FUNCTION_BLOCK LIntComparer EXTENDS Object IMPLEMENTS IComparer
VAR
	_ClassName : STRING := __POUNAME();
END_VAR

{attribute 'monitoring' := 'call'}
PROPERTY ClassName : STRING
GET
ClassName := _ClassName;
END_GET
END_PROPERTY

{attribute "object_name" := "Compare"}
METHOD Compare : COMPARISION_RESULT
VAR_INPUT
	left : __SYSTEM.AnyType;
	right : __SYSTEM.AnyType;
END_VAR
VAR
	leftPointer : POINTER TO LINT; 
	rightPointer : POINTER TO LINT; 
END_VAR
IF left.pValue = 0 AND right.pValue = 0 THEN
	Compare := COMPARISION_RESULT.FIRST_EQUAL_TO_SECOND;
	RETURN;
END_IF

IF left.pValue = 0 THEN
	Compare := COMPARISION_RESULT.FIRST_LESS_THAN_SECOND;
	RETURN;	
END_IF

IF right.pValue = 0 THEN
	Compare := COMPARISION_RESULT.FIRST_GREATER_THAN_SECOND;
	RETURN;	
END_IF

leftPointer := left.pValue;
rightPointer := right.pValue;

IF leftPointer^ < rightPointer^ THEN
	Compare := COMPARISION_RESULT.FIRST_LESS_THAN_SECOND;
ELSIF leftPointer^ > rightPointer^ THEN
	Compare := COMPARISION_RESULT.FIRST_GREATER_THAN_SECOND;
ELSE
	Compare := COMPARISION_RESULT.FIRST_EQUAL_TO_SECOND;	
END_IF
END_METHOD

{attribute 'monitoring' := 'call'}
PROPERTY Size : ULINT
GET
Size := XSIZEOF(THIS^);
END_GET
END_PROPERTY

END_FUNCTION_BLOCK

(* stored: Version 1.1.0.1
   POU LIntComparer: Id {6802d232-eb84-4fc6-9db7-da1a848885bb}, SpecialFunc None
   Property ClassName: Id {11696811-cbc8-4330-9b9c-34480612a1fd}
   Get Get: Id {9443910c-a564-4f25-a954-0af25c296bce}
   Method Compare: Id {16519cb2-8b2a-4d05-af51-ba14c0acf190}
   Property Size: Id {c25e4d6f-9f0f-4471-9ede-a23224e4040d}
   Get Get: Id {00ea876a-2583-4961-990c-bcb33b2f9770} *)
